// TIA Portal V17 export
// export: Created 2024-08-09T12:53:22.8235253Z, ExportSetting WithDefaults, DisplayName Totally Integrated Automation Portal, DisplayVersion V17 Update 7, DisplayName TIA Portal Openness, DisplayVersion V17 Update 7, DisplayName TIA Portal Version Control Interface, DisplayVersion V17, DisplayName STEP 7 Professional, DisplayVersion V17 Update 7, DisplayName STEP 7 Safety, DisplayVersion V17 Update 6, DisplayName WinCC Professional, DisplayVersion V17 Update 7
TYPE "S_ComLign"
// stored: IsFailsafeCompliant false
   STRUCT
      _PtcelOrig : "S_Cellule";   // cellule trouvee en table
      _Cases { ExternalAccessible := 'False'; ExternalVisible := 'False'; ExternalWritable := 'False'} : Array[0.."MAX_CASE"] of "S_Cases";
      _NoCommande { ExternalAccessible := 'False'; ExternalVisible := 'False'; ExternalWritable := 'False'} : String["T_COMM"];
      _NomClient { ExternalAccessible := 'False'; ExternalVisible := 'False'; ExternalWritable := 'False'} : String["T_CLIENT"];
      _Ville { ExternalAccessible := 'False'; ExternalVisible := 'False'; ExternalWritable := 'False'} : String["T_ADRESSE"];
      _CdMat { ExternalAccessible := 'False'; ExternalVisible := 'False'; ExternalWritable := 'False'} : String["T_CD_MAT"];
      _NoLot { ExternalAccessible := 'False'; ExternalVisible := 'False'; ExternalWritable := 'False'} : String["T_Num_Lot"];   // Numero de lot
      _LbMat { ExternalAccessible := 'False'; ExternalVisible := 'False'; ExternalWritable := 'False'} : String["T_LB_MAT"];
      _CdMatOrg { ExternalAccessible := 'False'; ExternalVisible := 'False'; ExternalWritable := 'False'} : String["T_CD_MAT"];
      _LbMatOrg { ExternalAccessible := 'False'; ExternalVisible := 'False'; ExternalWritable := 'False'} : String["T_LB_MAT"];
      _CdClient { ExternalAccessible := 'False'; ExternalVisible := 'False'; ExternalWritable := 'False'} : String;
      _Type { ExternalAccessible := 'False'; ExternalVisible := 'False'; ExternalWritable := 'False'} : Char;   // type de composant a charger P:Principal, M:Mineraux,R:Ratahce
      _QteChOrig : Real;
      _QteBrut : Real;   // quantite brut
      _QteTotComm { ExternalAccessible := 'False'; ExternalVisible := 'False'; ExternalWritable := 'False'} : Real;
      _QteTare : Real;   // poids tare dosage composant en kilos
      _QteDejaCharg : Real;
      _SeuilPV : Real;   // poids pour passage en PV
      _DebitCel { ExternalAccessible := 'False'; ExternalVisible := 'False'; ExternalWritable := 'False'} : Real;   // Debit cellule
      _TareCel { ExternalAccessible := 'False'; ExternalVisible := 'False'; ExternalWritable := 'False'} : Real;   // Tare composant cellule
      _QteNet : Real;   // poids Net
      _ConsArret : Real;   // Consigne d'arret
      _ConsQteTot : Real;   // poids a dosee pour la pesee
      _ChuteCel : Real;   // colonne de chute
      _Ecart : Real;   // Ecart dosage composant en kilos
      _Densite { ExternalAccessible := 'False'; ExternalVisible := 'False'; ExternalWritable := 'False'} : Real;   // densite produit
      _IdComLig { ExternalAccessible := 'False'; ExternalVisible := 'False'; ExternalWritable := 'False'} : ULInt;
      _IdLigOrig : ULInt;
      _VitGV : USInt;   // Vitesse variateur en GV
      _VitPV : USInt;   // Vitesse variateur en PV
      _NoLigne { ExternalAccessible := 'False'; ExternalVisible := 'False'; ExternalWritable := 'False'} : USInt;
      _NumPont { ExternalAccessible := 'False'; ExternalVisible := 'False'; ExternalWritable := 'False'} : USInt;   // Nom du pont de chargement utilise
      _Case { ExternalAccessible := 'False'; ExternalVisible := 'False'; ExternalWritable := 'False'} : USInt;
      _NmOrdre { ExternalAccessible := 'False'; ExternalVisible := 'False'; ExternalWritable := 'False'} : USInt;
      _NbCase { ExternalAccessible := 'False'; ExternalVisible := 'False'; ExternalWritable := 'False'} : USInt;
      _AutrePont { ExternalAccessible := 'False'; ExternalVisible := 'False'; ExternalWritable := 'False'} : Bool;   // fin du chargement sur autre pont
      _FgaVider { ExternalAccessible := 'False'; ExternalVisible := 'False'; ExternalWritable := 'False'} : Bool;   // flag de demande de vide cellule
   END_STRUCT;
END_TYPE
